(* CODESYS project zadatak4.project
   CustomField04_name: CustomField04
   CustomField06_name: CustomField06
   CustomField07_name: CustomField07
   CustomField09_name: CustomField09
   CustomField08_name: CustomField08
   CustomField02_name: CustomField02
   CustomField10_name: CustomField10
   CustomField01_name: CustomField01
   CustomField03_name: CustomField03
   CustomField05_name: CustomField05

Project tree, tasks and I/O mapping:
  MyController : TM238LFDC24DT, Schneider Electric, order no. TM238LFDC24DT, version 2.0.31.8
    application Application
      task MAST (cyclic, interval 20 ms, priority 15, watchdog 100 ms x 1) calls POU
      function HiddenPOU [ST]
      global variables GVL
      program POU [LD]
    CAN
    Embedded Functions
      PTO_PWM : PTO_PWM, Schneider Electric, version 2.0.31.8
        PTO_PWM
      HSC : HSC, Schneider Electric, version 2.0.31.8
        HSC
      IO : IO, Schneider Electric, version 2.0.31.8
          input  t2 : BOOL  // IW0.I9
          input  t1 : BOOL  // IW0.I10
          input  s1 : BOOL  // IW0.I11
          input  s2 : BOOL  // IW0.I12
          output z1 : BOOL  // QW0.Q4
          output zu1 : BOOL  // QW0.Q5
          output c1 : BOOL  // QW0.Q6
          output z2 : BOOL  // QW0.Q7
          output c2 : BOOL  // QW0.Q9
          unmapped channels: IW0, QW0
    Serial Line 2
      SoMachine_Network_Manager : SoMachine-Network_Manager, Schneider Electric, version 2.0.1.10
    Serial Line 1
      Modbus_Manager : Modbus_Manager, Schneider Electric, version 2.0.1.12
*)

// MyController/Application/GVL
VAR_GLOBAL
END_VAR

// MyController/Application/POU
PROGRAM POU
VAR
s1:BOOL;
s2:BOOL;
s3:BOOL;
s4:BOOL;
t1:BOOL;
t2:BOOL;
z1:BOOL;
zu1:BOOL;
c1:BOOL;
z2:BOOL;
c2:BOOL;
	sk1: BOOL;
	sk2: BOOL;
	b: BOOL;
	tp2: TP;
	c: BOOL;
	tp4: TP;
	ton1: TON;
	ton3: TON;
END_VAR
VAR // added by the converter: edge detectors and wires of the graphical bodies
    _w1, _w2, _w3, _w4, _w5, _w6 : BOOL;
END_VAR

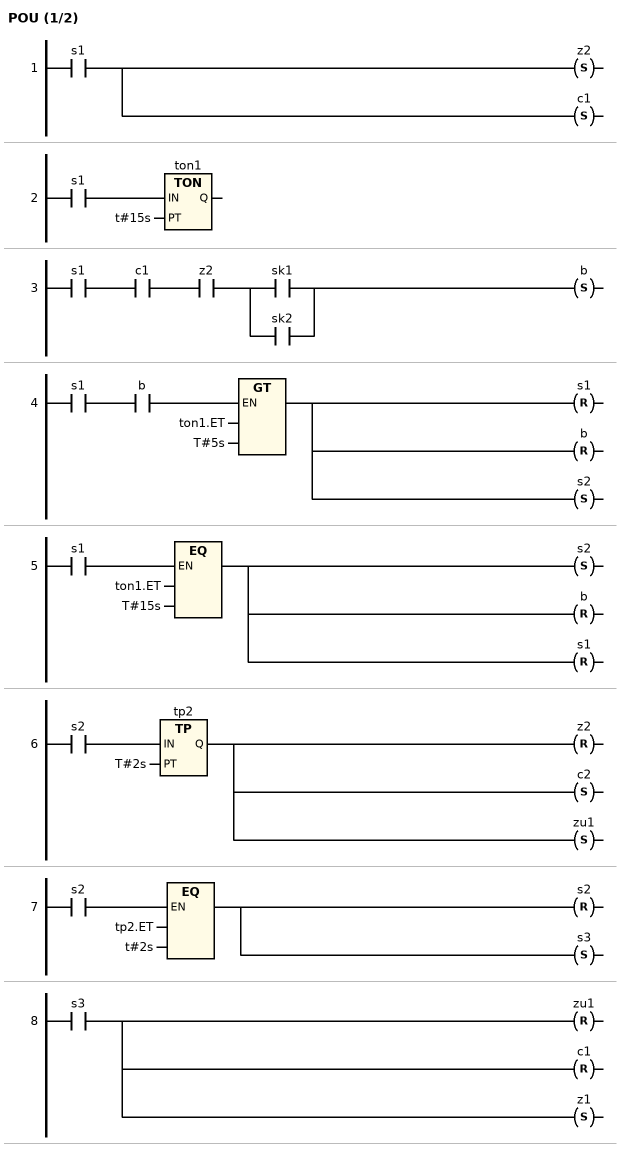
// NETWORK 1
z2 S= s1;
c1 S= s1;

// NETWORK 2
ton1(IN := s1, PT := t#15s); // TON

// NETWORK 3
b S= s1 AND c1 AND z2 AND (sk1 OR sk2);

// NETWORK 4
//   ton1.ET: elapsed time since rising edge at IN
_w1 := s1 AND b AND ton1.ET > T#5s;
s1 R= _w1;
b R= _w1;
s2 S= _w1;

// NETWORK 5
//   ton1.ET: elapsed time since rising edge at IN
_w2 := s1 AND ton1.ET = T#15s;
s2 S= _w2;
b R= _w2;
s1 R= _w2;

// NETWORK 6
tp2(IN := s2, PT := T#2s); // TP
z2 R= tp2.Q;
c2 S= tp2.Q;
zu1 S= tp2.Q;

// NETWORK 7
//   tp2.ET: elapsed time since pulse start
_w3 := s2 AND tp2.ET = t#2s;
s2 R= _w3;
s3 S= _w3;

// NETWORK 8
zu1 R= s3;
c1 R= s3;
z1 S= s3;

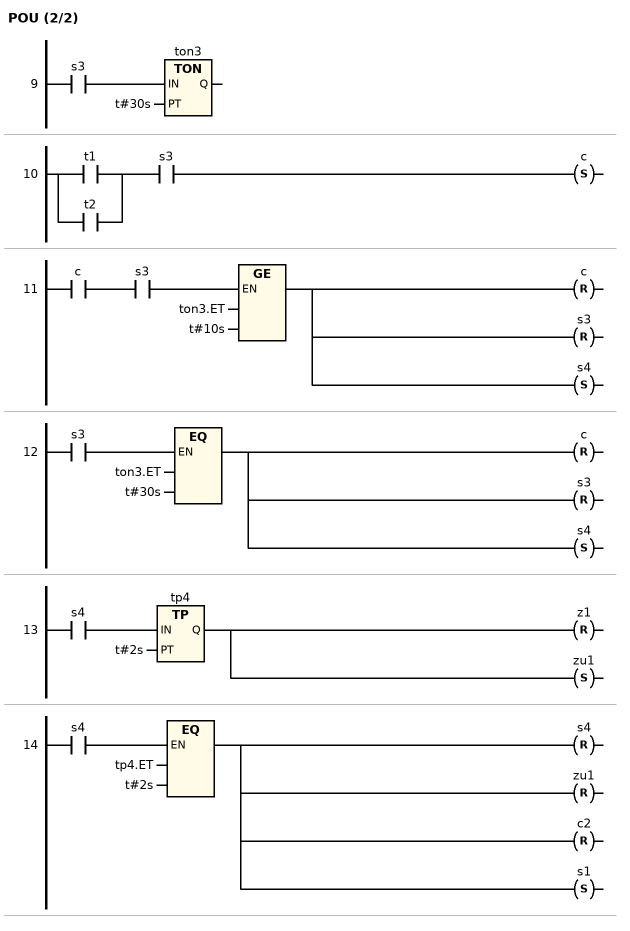
// NETWORK 9
ton3(IN := s3, PT := t#30s); // TON

// NETWORK 10
c S= (t1 OR t2) AND s3;

// NETWORK 11
//   ton3.ET: elapsed time since rising edge at IN
_w4 := c AND s3 AND ton3.ET >= t#10s;
c R= _w4;
s3 R= _w4;
s4 S= _w4;

// NETWORK 12
//   ton3.ET: elapsed time since rising edge at IN
_w5 := s3 AND ton3.ET = t#30s;
c R= _w5;
s3 R= _w5;
s4 S= _w5;

// NETWORK 13
tp4(IN := s4, PT := t#2s); // TP
z1 R= tp4.Q;
zu1 S= tp4.Q;

// NETWORK 14
//   tp4.ET: elapsed time since pulse start
_w6 := s4 AND tp4.ET = t#2s;
s4 R= _w6;
zu1 R= _w6;
c2 R= _w6;
s1 S= _w6;

END_PROGRAM

// MyController/Application/HiddenPOU
FUNCTION HiddenPOU : BOOL

VAR_INPUT
	pHiddenFunc: POINTER TO WORD;
END_VAR
VAR
	pRead: POINTER TO BYTE;
	pWrite: POINTER TO BYTE;
END_VAR

pRead := pHiddenFunc + 400;
pWrite := pHiddenFunc + 4400;
HiddenPOU := TRUE;

END_FUNCTION
